TYPE ST_PwrMgmt_HAWino_Out :
STRUCT
	bChargingActive					: BOOL;
	bExternalRecalibrationTrigger	: BOOL;
	fExternalRecalibrationValue		: LREAL;
	bComCheckRequest 				: BOOL;		// Request from charger to HAWino to test stable communication 
END_STRUCT 
END_TYPE

(* stored: Version 1.1.0.1, ProductVersion 3.1.4024.11
   DUT ST_PwrMgmt_HAWino_Out: Id {df863176-169d-4b16-be58-70303c30b253} *)
